FUNCTION_BLOCK FB_TelescopeMachine
VAR_INPUT
	bInit				: BOOL;
	bPark				: BOOL;
	bSlew				: BOOL;
	bTrack				: BOOL;
	bStop				: BOOL;
	bReset				: BOOL;
	
	fbParkedState		: I_TelescopeState;
	fbInitializingState	: I_TelescopeState;
	fbParkingState		: I_TelescopeState;
	fbIdleState			: I_TelescopeState;
	fbSlewingState		: I_TelescopeState;
	fbTrackingState		: I_TelescopeState;
	fbErrorState		: I_TelescopeState;
END_VAR
VAR_OUTPUT
	eState				: E_TelescopeState := E_TelescopeState.parked;
	ipState				: I_TelescopeState := fbParkedState;	
	eNextState			: E_TelescopeState;
END_VAR	
VAR	
	rtrigInit			: R_TRIG;
	rtrigPark			: R_TRIG;
	rtrigSlew			: R_TRIG;
	rtrigTrack			: R_TRIG;
	rtrigStop			: R_TRIG;
	rtrigReset			: R_TRIG;
	
	pControl 			: POINTER TO FB_BaseTelescopeControl;
END_VAR

rtrigInit(CLK := bInit);
rtrigPark(CLK := bPark);
rtrigSlew(CLK := bSlew);
rtrigTrack(CLK := bTrack);
rtrigStop(CLK := bStop);
rtrigReset(CLK := bReset);

IF rtrigInit.Q THEN
	ipState.Initialize();
END_IF

IF rtrigPark.Q THEN
	ipState.Park();
END_IF

IF rtrigSlew.Q THEN
	ipState.Slew(0, 0);
END_IF

IF rtrigTrack.Q THEN
	ipState.Track(0, 0);
END_IF

IF rtrigStop.Q THEN
	ipState.Stop();
END_IF

IF rtrigReset.Q THEN
	ipState.Reset();
END_IF

ipState.Main();

METHOD PRIVATE _GetState : I_TelescopeState
VAR_INPUT
	eState	: E_TelescopeState;
END_VAR
CASE State OF
	E_TelescopeState.parked:
		_GetState := fbParkedState;
	E_TelescopeState.initializing:
		_GetState := fbInitializingState;
	E_TelescopeState.parking:
		_GetState := fbParkingState;
	E_TelescopeState.idle:
		_GetState := fbIdleState;
	E_TelescopeState.slewing:
		_GetState := fbSlewingState;
	E_TelescopeState.tracking:
		_GetState := fbTrackingState;
END_CASE
END_METHOD

METHOD FB_init : BOOL
VAR_INPUT
	bInitRetains : BOOL; // if TRUE, the retain variables are initialized (warm start / cold start)
	bInCopyCode : BOOL;  // if TRUE, the instance afterwards gets moved into the copy code (online change)
	pControl : POINTER TO FB_BaseTelescopeControl;
END_VAR
THIS^.pControl := pControl;
END_METHOD

PROPERTY NextState : E_TelescopeState
GET
NextState := THIS^.eNextState;
END_GET
SET
THIS^.eNextState := NextState;
END_SET
END_PROPERTY

PROPERTY State : E_TelescopeState
GET
State := THIS^.eState;
END_GET
SET
THIS^.eState := State;
THIS^.ipState := THIS^._GetState(State);
THIS^.eNextState := E_TelescopeState.none;
END_SET
END_PROPERTY

END_FUNCTION_BLOCK

(* stored: Version 1.1.0.1, ProductVersion 3.1.4024.15
   POU FB_TelescopeMachine: Id {d878fe8e-6ab3-467d-9898-60a0958e8303}, SpecialFunc None
   Method _GetState: Id {7ec3eff3-6fdd-4614-9b7f-b2d995e8fb2c}
   Method FB_init: Id {3c22ef87-332a-4653-9eae-03a8b125faa1}
   Property NextState: Id {557174c8-f941-432c-856a-d20d0a114a36}
   Get Get: Id {6a1705a7-fc43-4f59-be74-ad0ef9f9ca86}
   Set Set: Id {ae4e4284-bc78-4249-99c5-85b5e1b1bf52}
   Property State: Id {8a257365-d0e0-49c6-ad50-1dc0f794a1fd}
   Get Get: Id {bac14e72-4e75-42fa-9d7d-04644d0b6712}
   Set Set: Id {ab3e2683-fe73-4c26-be05-bdf3f7bd2aee} *)
